FUNCTION_BLOCK ConveyorCTLRingToken (* Basic Function Block Type *)
  (* Standard: 61499-2 *)
  (* Version 0.2, 2003-12-04, JHC, Rockwell Automation, Renamed for better indexing. *)
  (* Version 0.1, 2002-11-05, JHC, Rockwell Automation, Corrected missing ST element in Algorithm REQ. *)
  (* Version 0.0, 2000-05-30, JHC, Rockwell Automation *)
  (* Compiler header: package fb.rt.cs725; *)
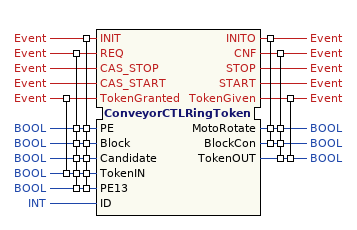
  EVENT_INPUT
    INIT WITH PE, Block, Candidate, TokenIN, PE13; (* Initialization Request *)
    REQ WITH PE, Block, Candidate, TokenIN, PE13; (* Normal Execution Request *)
    CAS_STOP;
    CAS_START;
    TokenGranted WITH TokenIN;
  END_EVENT
  EVENT_OUTPUT
    INITO WITH MotoRotate, BlockCon; (* Initialization Confirm *)
    CNF WITH MotoRotate, BlockCon, TokenOUT; (* Execution Confirmation *)
    STOP;
    START;
    TokenGiven WITH TokenOUT; (* Signal if Token Release or not *)
  END_EVENT
  VAR_INPUT
    PE : BOOL; (* Input event qualifier *)
    Block : BOOL;
    Candidate : BOOL;
    TokenIN : BOOL;
    PE13 : BOOL;
    ID : INT;
  END_VAR
  VAR_OUTPUT
    MotoRotate : BOOL; (* Output event qualifier *)
    BlockCon : BOOL;
    TokenOUT : BOOL;
  END_VAR
  VAR
    lastPE : BOOL := 1;
    lastBlock : BOOL := 0;
  END_VAR
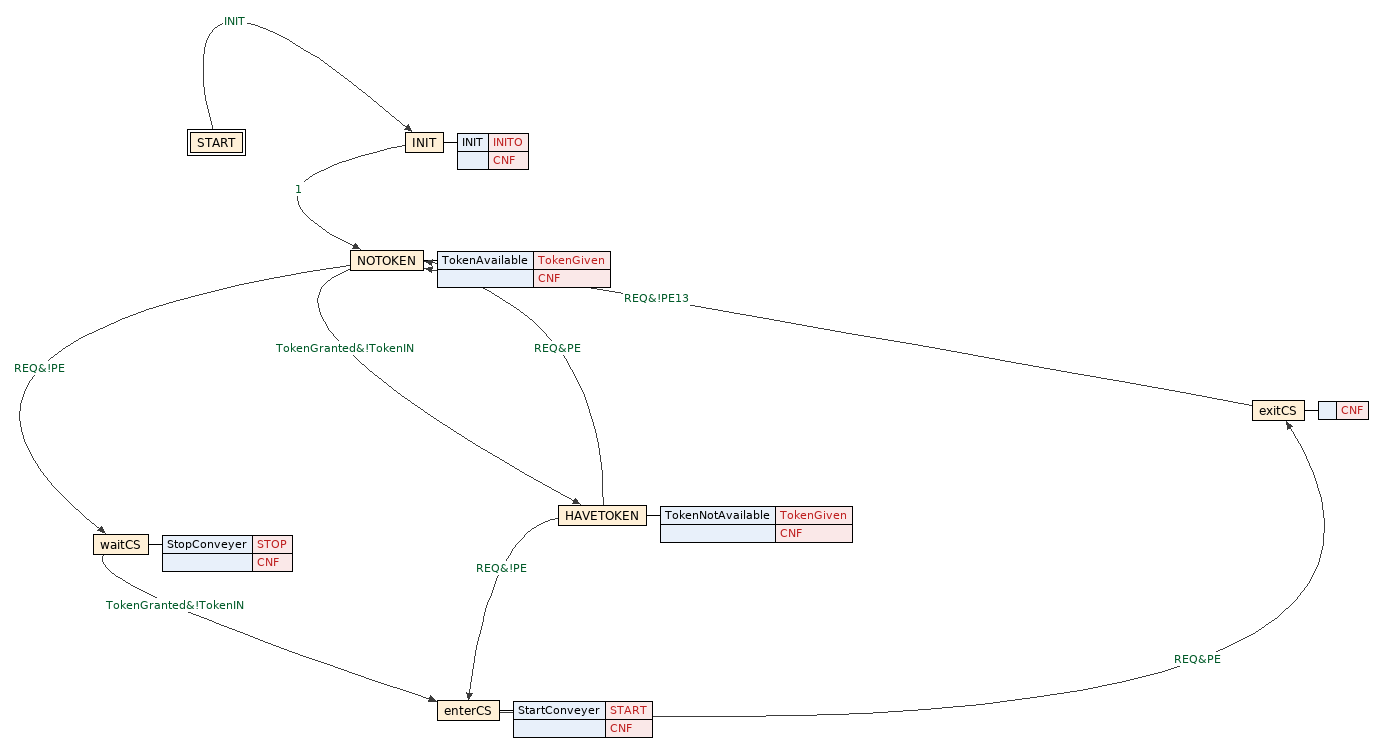
  EC_STATES
    START; (* Initial State *)
    INIT : INIT -> INITO, -> CNF; (* Initialization *)
    NOTOKEN : TokenAvailable -> TokenGiven, -> CNF;
    waitCS : StopConveyer -> STOP, -> CNF; (* waiting to enter critical section *)
    HAVETOKEN : TokenNotAvailable -> TokenGiven, -> CNF;
    enterCS : StartConveyer -> START, -> CNF;
    exitCS : -> CNF;
  END_STATES
  EC_TRANSITIONS
    START TO INIT := INIT;
    INIT TO NOTOKEN := 1;
    NOTOKEN TO waitCS := REQ&!PE; (* When we want to enter the section *)
    NOTOKEN TO HAVETOKEN := TokenGranted&!TokenIN; (* Other token is granting access *)
    HAVETOKEN TO NOTOKEN := REQ&PE; (* Have the token but dont want to use critical section *)
    waitCS TO enterCS := TokenGranted&!TokenIN; (* Other process is giving access *)
    HAVETOKEN TO enterCS := REQ&!PE; (* The process wants to enter critical section *)
    enterCS TO exitCS := REQ&PE; (* All items waiting go through *)
    exitCS TO NOTOKEN := REQ&!PE13;
  END_TRANSITIONS
  ALGORITHM INIT IN ST: (* Initialization algorithm *)
MotoRotate := TRUE;
Block := FALSE;

System.out.println(this + " " + MotoRotate);
System.out.println(MotoRotate);
  END_ALGORITHM
  ALGORITHM REQ IN ST: (* Normally executed algorithm *)
System.out.println(this +  " -> Candidate" + Candidate);
IF Candidate THEN
IF lastPE !:= PE THEN
IF NOT PE THEN
BlockCon:= TRUE;
System.out.println("BlockCon = true");
ELSE
BlockCon:=FALSE;
System.out.println("BlockCon = false");
END_IF
lastPE := PE;
END_IF
IF lastBlock !:= Block THEN
IF Block THEN
STOP.serviceEvent(this);
MotoRotate := FALSE;
System.out.println("Cas Stop");
ELSE
START.serviceEvent(this);
MotoRotate := TRUE;
System.out.println("Cas Start");
END_IF
lastBlock := Block;
END_IF
END_IF
  END_ALGORITHM
  ALGORITHM START IN ST:
MotoRotate:=TRUE;
System.out.println(this + " Start " + MotoRotate);

System.out.println("Start " + MotoRotate);
  END_ALGORITHM
  ALGORITHM STOP IN ST:
MotoRotate := FALSE;
System.out.println(this + " Stop " + MotoRotate);

System.out.println("Stop " + MotoRotate);
  END_ALGORITHM
  ALGORITHM TokenAvailable IN Java: (* Free the token since we are not using it. *)
System.out.println(ID.value +"No Token");
TokenOUT.value = false;
  END_ALGORITHM
  ALGORITHM StopConveyer IN Java:
BlockCon.value = true;
System.out.println(ID.value +"Wait CS");
MotoRotate.value = false;
  END_ALGORITHM
  ALGORITHM TokenNotAvailable IN Java: (* Tell the other processes we are using the token *)
System.out.println(ID.value +"Have Token");
TokenOUT.value = true;
  END_ALGORITHM
  ALGORITHM StartConveyer IN Java: (* Start the conveyer as we are entering critical section *)
BlockCon.value = false;
MotoRotate.value = true;
System.out.println(ID.value +"Start Conveyer");
  END_ALGORITHM
END_FUNCTION_BLOCK
